// TIA Portal V20 export
DATA_BLOCK "HmiInterface"   // DB96
{ DB_Accessible_From_OPC_UA := 'FALSE' }
AUTHOR : ERsystem_FA2_DH. Kim
// stored: Access Published, DBAccessibleFromOPCUA false, DBAccessibleFromWebserver false, MemoryReserve 100, Namespace Unit1.Em1
   VAR
      em : "LAF_typeEmInterface";
      cm : Struct
         softCam : "Unit1.type_emRelations_em1_SoftCam";
         brakeTest : Struct
            UnwinderBtmAxisB : "LER_typeBrakeTestEmInterface";
         END_STRUCT;
      END_STRUCT;
      sepaUnwinderBtm : Struct
         jobs { S7_SetPoint := 'True'} : "LAF_typeJobsInterface";
         sequence { S7_SetPoint := 'True'} : "LAF_typeSequenceInterface";
      END_STRUCT;
      auxiliary : Struct
         cmEpc_UnUse : Bool;
         AutoSpliceRemainingLength : LReal;
      END_STRUCT;
      cmBtmDirectionCheckSensor { S7_SetPoint := 'True'} : "LBC_typeDigitalSignalInterface";
      cmRadiusMeasureBtm : "LBC_typeAnalogInputInterface";
   END_VAR
   VAR RETAIN
      cmRadiusMeasure : "LER_typeRadiusMeasureInterface";
   END_VAR
   VAR
      cmUnwinderBtmAxisB : "LBC_typeAxis64PosInterface";
      cmAirShaftBtmOnOff : "LBC_typeTwoWayActuatorInterface";
      cmEpcBtm : "LER_typeCON600Interface";
      motion : Struct
         jobs { S7_SetPoint := 'True'} : "LAF_typeJobsInterface";
         sequence { S7_SetPoint := 'True'} : "LAF_typeSequenceInterface";
      END_STRUCT;
      "step" : Struct
         jobs { S7_SetPoint := 'True'} : "LAF_typeJobsInterface";
         sequence { S7_SetPoint := 'True'} : "LAF_typeSequenceInterface";
      END_STRUCT;
      intCondition : Struct
         Axis_02 { S7_SetPoint := 'True'} : "LER.typeAxisIntlockAll";   // UnwinderBottomAxisB
         Actuator_02 { S7_SetPoint := 'True'} : "LER.typeAxisActuatorCondition";   // UnwinderAirShaftBottom
      END_STRUCT;
   END_VAR
BEGIN
   em.interlinkMode.link := FALSE;
   em.interlinkMode.unlink := FALSE;
   em.interlinkMode.isLinked := TRUE;
   em.commands.enable := FALSE;
   em.commands.acknowledge := FALSE;
   em.commands.disableAlarms := FALSE;
   em.commands.activateSimulation := FALSE;
   em.commands.home := FALSE;
   em.commands.moveToInitialPosition := FALSE;
   em.commands.directModeControl := 16#0000_0002;
   em.commands.directStateControl := 16#0000_0002;
   em.status.enabled := TRUE;
   em.status.acknowledgeActive := FALSE;
   em.status.alarmsDisabled := FALSE;
   em.status.simulationActive := FALSE;
   em.status.safetyReleased := TRUE;
   em.status.initialized := FALSE;
   em.status.homed := FALSE;
   em.status.safeState := TRUE;
   em.status.stateComplete := TRUE;
   cmBtmDirectionCheckSensor.commands.refreshConfiguration := FALSE;
   cmBtmDirectionCheckSensor.commands.editConfiguration := FALSE;
   cmBtmDirectionCheckSensor.commands.saveConfiguration := FALSE;
   cmBtmDirectionCheckSensor.commands.reset := FALSE;
   cmBtmDirectionCheckSensor.monitoring.enable := TRUE;
   cmBtmDirectionCheckSensor.monitoring.referenceDesignator := WSTRING#'U1.EM1 SepaUnwinderBtm.cmBtmDirectionCheckSensor';
   cmBtmDirectionCheckSensor.monitoring.simulation := FALSE;
   cmBtmDirectionCheckSensor.monitoring.processValue := TRUE;
   cmBtmDirectionCheckSensor.monitoring.error := FALSE;
   cmBtmDirectionCheckSensor.monitoring.status := 16#0000;
   cmBtmDirectionCheckSensor.configuration.referenceDesignator := WSTRING#'cmBtmDirectionCheckSensor';
   cmBtmDirectionCheckSensor.configuration.onDelay := T#0MS;
   cmBtmDirectionCheckSensor.configuration.offDelay := T#0MS;
   cmBtmDirectionCheckSensor.configuration.default := FALSE;
   cmBtmDirectionCheckSensor.configuration.invertProcessValue := FALSE;
   cmBtmDirectionCheckSensor.configuration.disableAlarms := FALSE;
   cmRadiusMeasureBtm.commands.refreshConfiguration := FALSE;
   cmRadiusMeasureBtm.commands.editConfiguration := FALSE;
   cmRadiusMeasureBtm.commands.saveConfiguration := FALSE;
   cmRadiusMeasureBtm.commands.reset := FALSE;
   cmRadiusMeasureBtm.monitoring.enable := TRUE;
   cmRadiusMeasureBtm.monitoring.referenceDesignator := WSTRING#'U1.EM1 SepaUnwinderBtm.cmRadiusMeasureBtm';
   cmRadiusMeasureBtm.monitoring.simulation := FALSE;
   cmRadiusMeasureBtm.monitoring.processValue := 0.0;
   cmRadiusMeasureBtm.monitoring.analogValue := -4864;
   cmRadiusMeasureBtm.monitoring.limitHigh2 := FALSE;
   cmRadiusMeasureBtm.monitoring.limitHigh1 := FALSE;
   cmRadiusMeasureBtm.monitoring.limitLow1 := TRUE;
   cmRadiusMeasureBtm.monitoring.limitLow2 := TRUE;
   cmRadiusMeasureBtm.monitoring.maxValueReached := FALSE;
   cmRadiusMeasureBtm.monitoring.minValueReached := TRUE;
   cmRadiusMeasureBtm.monitoring.error := TRUE;
   cmRadiusMeasureBtm.monitoring.status := 16#8405;
   cmRadiusMeasureBtm.configuration.referenceDesignator := WSTRING#'cmRadiusMeasureBtm';
   cmRadiusMeasureBtm.configuration.physicalUnit := 'unit';
   cmRadiusMeasureBtm.configuration.isUnipolarSignal := TRUE;
   cmRadiusMeasureBtm.configuration.default := 0.0;
   cmRadiusMeasureBtm.configuration.limitHigh2 := 400.0;
   cmRadiusMeasureBtm.configuration.limitHigh1 := 400.0;
   cmRadiusMeasureBtm.configuration.limitLow1 := 0.0;
   cmRadiusMeasureBtm.configuration.limitLow2 := 0.0;
   cmRadiusMeasureBtm.configuration.processValueMax := 400.0;
   cmRadiusMeasureBtm.configuration.processValueMin := 0.0;
   cmRadiusMeasureBtm.configuration.scaleAnalogUppPoint := 27648.0;
   cmRadiusMeasureBtm.configuration.scaleAnalogLowPoint := 0.0;
   cmRadiusMeasureBtm.configuration.scaleProcessUppPoint := 400.0;
   cmRadiusMeasureBtm.configuration.scaleProcessLowPoint := 0.0;
   cmRadiusMeasureBtm.configuration.disableAlarms := TRUE;
   cmRadiusMeasure.commands.ZeroSet := FALSE;
   cmRadiusMeasure.commands.Reset := FALSE;
   cmRadiusMeasure.monitoring.Radius := 36.0;
   cmRadiusMeasure.monitoring.Diameter := 72.0;
   cmRadiusMeasure.configuration.Offset := 0.0;
   cmRadiusMeasure.configuration.DecimalPoint := 0;
   cmAirShaftBtmOnOff.commands.refreshConfiguration := FALSE;
   cmAirShaftBtmOnOff.commands.editConfiguration := FALSE;
   cmAirShaftBtmOnOff.commands.saveConfiguration := FALSE;
   cmAirShaftBtmOnOff.commands.reset := FALSE;
   cmAirShaftBtmOnOff.commands.commandHomePos := FALSE;
   cmAirShaftBtmOnOff.commands.commandWorkPos := FALSE;
   cmAirShaftBtmOnOff.monitoring.enable := TRUE;
   cmAirShaftBtmOnOff.monitoring.referenceDesignator := WSTRING#'U1.EM1 SepaUnwinderBtm.cmAirShaftBtmOnOff';
   cmAirShaftBtmOnOff.monitoring.commandHomePos := FALSE;
   cmAirShaftBtmOnOff.monitoring.commandWorkPos := FALSE;
   cmAirShaftBtmOnOff.monitoring.goToHomePos := FALSE;
   cmAirShaftBtmOnOff.monitoring.goToWorkPos := FALSE;
   cmAirShaftBtmOnOff.monitoring.inHomePos := FALSE;
   cmAirShaftBtmOnOff.monitoring.inWorkPos := FALSE;
   cmAirShaftBtmOnOff.monitoring.reset := FALSE;
   cmAirShaftBtmOnOff.monitoring.enableManualCmds := TRUE;
   cmAirShaftBtmOnOff.monitoring.error := FALSE;
   cmAirShaftBtmOnOff.monitoring.interlockHomePos := TRUE;
   cmAirShaftBtmOnOff.monitoring.interlockWorkPos := TRUE;
   cmAirShaftBtmOnOff.monitoring.status := 16#7003;
   cmAirShaftBtmOnOff.monitoring.interlockWarningWorkPos := FALSE;
   cmAirShaftBtmOnOff.monitoring.interlockWarningHomePos := FALSE;
   cmAirShaftBtmOnOff.configuration.referenceDesignator := WSTRING#'cmAirShaftBtmOnOff';
   cmAirShaftBtmOnOff.configuration.monitoringLeavingFeedback := T#5S;
   cmAirShaftBtmOnOff.configuration.monitoringReachingFeedback := T#5S;
   cmAirShaftBtmOnOff.configuration.monitoringDiscrepancy := T#0MS;
   cmAirShaftBtmOnOff.configuration.setOutputHomeContinuously := TRUE;
   cmAirShaftBtmOnOff.configuration.setOutputWorkContinuously := TRUE;
   cmAirShaftBtmOnOff.configuration.disableHomeCommand := FALSE;
   cmAirShaftBtmOnOff.configuration.disableFeedbackHomePos := FALSE;
   cmAirShaftBtmOnOff.configuration.disableFeedbackWorkPos := FALSE;
   cmAirShaftBtmOnOff.configuration.disableAlarms := FALSE;
   cmAirShaftBtmOnOff.configuration.resetOutputsOnError := FALSE;
   cmAirShaftBtmOnOff.configuration.allwaysWaitOnReachingTime := FALSE;
END_DATA_BLOCK
